{attribute 'linkalways'} 
{attribute 'no_explicit_call' := 'This FB is a CLASS and must be accessed using methods or properties'}
{attribute 'enable_dynamic_creation'}
FUNCTION_BLOCK _ETcVnVectorCompareMethod EXTENDS EnumDatatypeBase
VAR
	localData : ETcVnVectorCompareMethod;
	activeData : REFERENCE TO ETcVnVectorCompareMethod;
	enumBaseDatatype : _DINT(localData);
END_VAR

METHOD PRIVATE AddLocalEnumeration
VAR_INPUT
	Enumeration : T_MAXSTRING;
	Value : ETcVnVectorCompareMethod;
END_VAR
AddEnumeration(Enumeration, Value);
END_METHOD

PROPERTY PUBLIC Address : PVOID
GET
Address := ADR(activeData);
END_GET
END_PROPERTY

METHOD PUBLIC ClearReference
VAR_INPUT
END_VAR
activeData REF= localData;
SetBaseDatatypeReference();
END_METHOD

METHOD PUBLIC Clone : I_Datatype
VAR
    pClone : POINTER TO _ETcVnVectorCompareMethod;
END_VAR
pClone := __NEW(_ETcVnVectorCompareMethod(InitialValue := Value));
Clone := pClone^;
END_METHOD

METHOD FB_init : BOOL
VAR_INPUT
	bInitRetains : BOOL; // if TRUE, the retain variables are initialized (warm start / cold start)
	bInCopyCode : BOOL;  // if TRUE, the instance afterwards gets moved into the copy code (online change)
	InitialValue : ETcVnVectorCompareMethod;
END_VAR
localData := InitialValue;
AddBaseDatatype(enumBaseDatatype);
ClearReference();

AddLocalEnumeration('TCVN_VCM_EUCLIDEAN', ETcVnVectorCompareMethod.TCVN_VCM_EUCLIDEAN);
AddLocalEnumeration('TCVN_VCM_ELEMENTWISE', ETcVnVectorCompareMethod.TCVN_VCM_ELEMENTWISE);
END_METHOD

PROPERTY PUBLIC Identifier : T_MAXSTRING
GET
Identifier := 'ETcVnVectorCompareMethod';
END_GET
END_PROPERTY

METHOD IsEnumeratorValueEqual : BOOL
VAR_INPUT
	Enumerator : I_KeyValueForwardEnumerator;
END_VAR
VAR
	storedValue : ETcVnVectorCompareMethod;
END_VAR
IF NOT Enumerator.TryGet(storedValue) THEN
	RETURN;
END_IF

IsEnumeratorValueEqual := storedValue = activeData;
END_METHOD

METHOD PUBLIC MakeReferenceTo
VAR_INPUT
	ReferenceTarget : REFERENCE TO ETcVnVectorCompareMethod;
END_VAR
activeData REF= ReferenceTarget;
SetBaseDatatypeReference();
END_METHOD

METHOD PROTECTED SetBaseDatatypeReference
VAR_INPUT
END_VAR
enumBaseDatatype.MakeReferenceTo(activeData);
END_METHOD

PROPERTY PUBLIC Size : UDINT
GET
Size := SIZEOF(activeData);
END_GET
END_PROPERTY

METHOD TryMakeReferenceTo : BOOL
VAR_INPUT
	Target : I_Datatype;
END_VAR
VAR
	targetAsEnum : I_EnumDatatype;
	pTargetData : POINTER TO ETcVnVectorCompareMethod;
END_VAR
IF NOT Target.TryResolveAsEnumDatatype(targetAsEnum) THEN
	RETURN;
END_IF

IF targetAsEnum.Identifier <> Identifier THEN
	RETURN;
END_IF

pTargetData := Target.Address;
activeData REF= pTargetData^;
SetBaseDatatypeReference();
TryMakeReferenceTo := TRUE;
END_METHOD

PROPERTY PUBLIC Value : ETcVnVectorCompareMethod
GET
Value := activeData;
END_GET
SET
activeData := Value;
END_SET
END_PROPERTY

END_FUNCTION_BLOCK

(* stored: Version 1.1.0.1
   POU _ETcVnVectorCompareMethod: Id {b8fea9f0-05f1-4a93-a190-384c4e52fa47}, SpecialFunc None
   Folder Constructor: Id {e3b4ff00-84a5-4135-91b0-511c5d8b631b}
   Folder Private: Id {9f7e37e4-e517-4343-ac79-c32a9eea6e6e}
   Folder Protected: Id {b18b4e9b-076a-4833-a007-6d44ce6085a6}
   Method AddLocalEnumeration: Id {58b13a54-f95d-4c6b-a4de-b0da329ab6f3}
   Property Address: Id {21065c53-8d5c-47ba-be81-6e18ef373feb}
   Get Get: Id {ecf655a8-4e91-4733-86bc-6c4e74cbc99a}
   Method ClearReference: Id {92ca6c39-bbdb-4fb2-8d00-aee6ed2fc572}
   Method Clone: Id {a0045089-a652-408e-a4c8-2310870e1864}
   Method FB_init: Id {d370d360-d9bc-4005-bea2-1af4172745e3}
   Property Identifier: Id {a07b20da-77eb-4fbf-a45e-875a4e49bb89}
   Get Get: Id {cba60229-ecf9-4827-bf91-24be20c3ba5d}
   Method IsEnumeratorValueEqual: Id {783a1fbe-4e82-47f8-8334-3764c9fba1ec}
   Method MakeReferenceTo: Id {8bcbb42c-0c7f-4350-a87e-8c8340baacab}
   Method SetBaseDatatypeReference: Id {e69613fd-0acc-4b04-9682-28631f6350e9}
   Property Size: Id {46c1b6c4-6927-4dc9-bb3f-f29023648638}
   Get Get: Id {5b7bdc62-015f-46f3-8606-9e5097280a33}
   Method TryMakeReferenceTo: Id {aaa7ea6c-1728-4060-bcd1-2365b0d3bf34}
   Property Value: Id {96a1899d-a0b5-449a-b1e7-b763249dad75}
   Get Get: Id {f451bcd3-5404-4a74-a79e-67d94283423f}
   Set Set: Id {1bf8df7a-d90a-4258-a614-15b4b92b6e46} *)
